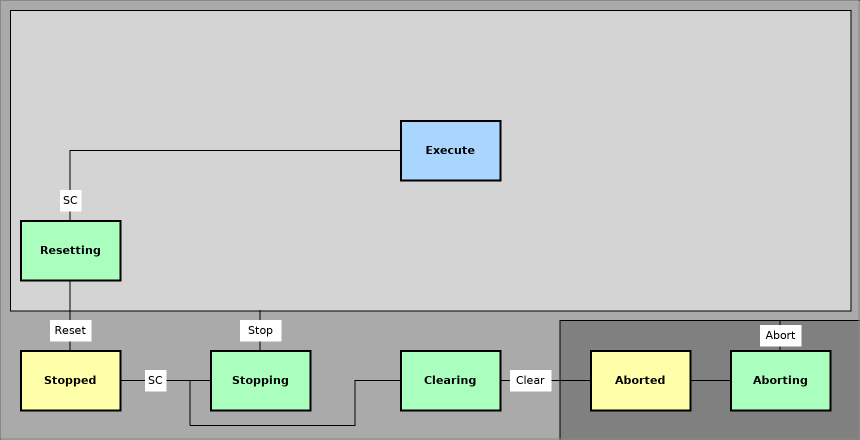
VISUALIZATION VFM_PackML_Manual  // 860x440
VAR_IN_OUT
	HMI : ST_PackMLBaseModule_HMI;
END_VAR
    Rectangle (560,320 301x121)
    Rectangle (10,10 841x301)
    Rectangle (590,350 101x61), "Aborted", colour toggle: HMI.Status.State = Tc3_PackML_V2.E_PMLState.ePMLState_Aborted
    Rectangle (400,350 101x61), "Clearing", colour toggle: HMI.Status.State = Tc3_PackML_V2.E_PMLState.ePMLState_Clearing
    Rectangle (210,350 101x61), "Stopping", colour toggle: HMI.Status.State = Tc3_PackML_V2.E_PMLState.ePMLState_Stopping
    Rectangle (20,350 101x61), "Stopped", colour toggle: HMI.Status.State = Tc3_PackML_V2.E_PMLState.ePMLState_Stopped
    Rectangle (20,220 101x61), "Resetting", colour toggle: HMI.Status.State = Tc3_PackML_V2.E_PMLState.ePMLState_Resetting
    Rectangle (400,120 101x61), "Execute", colour toggle: HMI.Status.State = Tc3_PackML_V2.E_PMLState.ePMLState_Execute
    Rectangle (730,350 101x61), "Aborting", colour toggle: HMI.Status.State = Tc3_PackML_V2.E_PMLState.ePMLState_Aborting
    Line (0,0) (860,0)
    Line (860,0) (860,320)
    Line (560,320) (860,320)
    Line (560,440) (560,320)
    Line (0,440) (560,440)
    Line (0,440) (0,0)
    Line (780,350) (780,320)
    Line (690,380) (730,380)
    Line (355,380) (400,380)
    Line (500,380) (590,380)
    Line (355,425) (355,380)
    Line (190,425) (355,425)
    Line (260,350) (260,310)
    Line (120,380) (210,380)
    Line (70,150) (400,150)
    Line (190,425) (190,380)
    Line (70,350) (70,280)
    Line (70,220) (70,150)
    Rectangle (760,325 41x21), "Abort"
    Rectangle (50,320 41x21), "Reset"
    Rectangle (510,370 41x21), "Clear"
    Rectangle (240,320 41x21), "Stop"
    Rectangle (145,370 21x21), "SC"
    Rectangle (60,190 21x21), "SC"
END_VISUALIZATION

(* stored: Version 1.1.0.1, ProductVersion 3.1.4024.12
   Visu VFM_PackML_Manual: Id {6085f019-4672-466c-95da-ff947730e40b} *)
